Yaskawa INFORM job: R1_W49-52-A1(90,180)KM-OK.JBI

/JOB
//NAME R1_W49-52-A1(90,180)KM-OK
///FOLDERNAME KRIS-SCIANA
//POS
///NPOS 79,79,0,5,0,0
///TOOL 0
///POSTYPE PULSE
///PULSE
C00000=109471,-80411,-71829,-33263,113126,21380
C00001=-48619,-15555,-18243,-18279,95335,-12517
C00002=-74776,32390,22089,-16092,92623,-17270
C00003=-74867,35757,29537,-16050,89859,-16941
C00004=-75036,36599,32361,-16047,88568,-16832
C00005=-75036,36895,33395,-16047,88102,-16772
C00006=-74903,37254,32698,-16044,88719,-16805
C00007=-72459,12362,8558,-16008,91190,-16266
C00008=-61209,-17232,-1681,-36622,66784,-6421
C00009=-61731,-16191,-908,-36534,66611,-6591
C00010=-59990,-21702,-9204,-36261,69196,-6738
C00011=-72720,3761,1433,-15340,81732,-21663
C00012=-72610,7758,8804,-15444,79356,-21325
C00013=-73045,10828,13692,-15468,77892,-21294
C00014=-73045,10997,14245,-15480,77647,-21262
C00015=-73045,10828,13692,-15468,77892,-21294
C00016=-72048,12642,15323,-15567,78014,-20955
C00017=-73045,10828,13692,-15468,77892,-21294
C00018=-79642,10121,9779,-4752,79820,-25647
C00019=-80358,6534,2777,-4651,82236,-25983
C00020=-69953,-20577,-2415,-29105,71989,2082
C00021=-71388,-15105,4995,-29275,69960,2047
C00022=-71943,-12839,8075,-29360,69127,2048
C00023=-71949,-11985,10076,-29503,68430,2234
C00024=-71943,-12839,8075,-29360,69127,2048
C00025=-78156,-21778,1298,-21120,59983,-2481
C00026=-78744,-20042,2543,-20963,59953,-2712
C00027=-78156,-21778,1298,-21120,59983,-2481
C00028=-77865,-24315,-1842,-21059,60645,-2495
C00029=-77104,-30529,-9436,-20946,62223,-2499
C00030=-66753,-24791,-5212,-33273,69818,4262
C00031=-68453,-19258,1867,-33429,67885,4157
C00032=-69108,-16977,4805,-33509,67096,4131
C00033=-69405,-16270,5329,-33473,67016,4031
C00034=-69412,-15422,7310,-33651,66355,4242
C00035=-69405,-16270,5329,-33473,67016,4031
C00036=-69108,-16977,4805,-33509,67096,4131
C00037=-78682,-30038,-3543,-25118,55124,-1302
C00038=-79303,-28327,-2398,-24897,55100,-1566
C00039=-78682,-30038,-3543,-25118,55124,-1302
C00040=-75986,-28450,-4438,-25449,57169,-654
C00041=-75599,-31023,-7408,-25413,57744,-634
C00042=-74583,-37366,-14608,-25368,59113,-542
C00043=-54832,-34796,3895,-72693,39731,-39244
C00044=-56965,-32089,5608,-72268,38461,-39820
C00045=-57882,-31468,9455,-80412,35987,-35279
C00046=-57943,-31847,4343,-71137,38137,-40613
C00047=-56828,-32279,5486,-72299,38543,-39782
C00048=-56494,-29260,14044,-87349,37133,-31586
C00049=-56951,-32108,5596,-72272,38470,-39816
C00050=-54817,-34814,3883,-72695,39739,-39240
C00051=-70512,18761,16215,-24928,63616,-33333
C00052=-71276,21755,18910,-24702,63280,-33571
C00053=-71200,18616,16875,-24804,62971,-33467
C00054=-70825,17807,14425,-24705,64080,-33568
C00055=-67366,10962,9433,-25880,64732,-32303
C00056=-67541,9161,7476,-25769,64930,-32423
C00057=-66799,6994,5573,-25983,65214,-32188
C00058=-71450,3986,10861,-16686,71001,-58886
C00059=-83506,38901,46150,-14860,73867,-63488
C00060=-83557,40717,50113,-14966,72402,-63324
C00061=-72489,19688,28494,-17099,68495,19316
C00062=-72729,20279,28486,-17025,68740,19190
C00063=-86229,35527,44055,-7657,69598,-64559
C00064=-83557,39592,48403,-4091,67286,-63785
C00065=-82033,27096,36992,-6435,61524,-62871
C00066=-80468,765,21137,-10528,40199,-59994
C00067=-83053,-10240,21848,-3806,20837,-60444
C00068=-83052,-10243,21845,-3807,20837,-60443
C00069=-68410,-14368,18791,-25286,23146,-48376
C00070=-67879,-14666,18605,-25978,23265,-47975
C00071=-67391,-14563,19188,-26892,23140,-47472
C00072=-67758,-15818,19043,-27038,22532,-47449
C00073=-67911,-23908,2369,-21552,28082,-50172
C00074=-67911,-23908,2369,-21552,28082,-50172
C00075=-73405,-104993,-53637,-20388,20000,-51360
C00076=-27978,-168994,-134866,-21563,-5876,-50681
C00077=15433,-168994,-134866,-21563,-5876,-50681
C00078=15433,-168994,-134866,-21563,-5876,-50681
BC00000=66192,1897,868014
BC00001=55231,1826,395730
BC00002=53649,1816,327568
BC00003=53649,1816,327568
BC00004=53649,1816,327568
BC00005=53649,1816,327568
BC00006=53649,1816,327568
BC00007=53649,1816,327568
BC00008=53649,1816,327568
BC00009=53649,1816,327568
BC00010=53649,1816,327568
BC00011=81522,15,359812
BC00012=81522,15,359812
BC00013=81522,15,359812
BC00014=81522,15,359812
BC00015=81522,15,359812
BC00016=81522,15,359812
BC00017=81522,15,359812
BC00018=81522,15,359812
BC00019=81522,15,359812
BC00020=119220,15,404761
BC00021=119220,15,404761
BC00022=119220,15,404761
BC00023=119220,15,404761
BC00024=119220,15,404761
BC00025=119220,15,404761
BC00026=119220,15,404761
BC00027=119220,15,404761
BC00028=119220,15,404761
BC00029=119220,15,404761
BC00030=91379,15,388853
BC00031=91379,15,388853
BC00032=91379,15,388853
BC00033=91379,15,388853
BC00034=91379,15,388853
BC00035=91379,15,388853
BC00036=91379,15,388853
BC00037=91379,15,388853
BC00038=91379,15,388853
BC00039=91379,15,388853
BC00040=91379,15,388853
BC00041=91379,15,388853
BC00042=91379,15,388853
BC00043=52539,15,360662
BC00044=53193,15,340173
BC00045=53455,15,331978
BC00046=53455,15,331978
BC00047=53455,15,331978
BC00048=85993,15,331095
BC00049=85731,15,339290
BC00050=85076,15,359778
BC00051=28900,15,309803
BC00052=29839,15,300407
BC00053=29839,15,300407
BC00054=29839,15,300407
BC00055=36980,15,283561
BC00056=36041,15,292958
BC00057=33695,15,316449
BC00058=58127,15,406832
BC00059=58127,15,406832
BC00060=58127,15,406832
BC00061=57102,15,378985
BC00062=57102,15,378985
BC00063=58127,15,406832
BC00064=58127,15,406832
BC00065=58127,15,406832
BC00066=58127,15,406832
BC00067=58127,15,406831
BC00068=58127,15,406831
BC00069=58127,15,406831
BC00070=58127,15,406831
BC00071=58127,15,406831
BC00072=58127,15,406831
BC00073=58127,15,406831
BC00074=58127,15,406831
BC00075=58127,15,406831
BC00076=8067,559,1056049
BC00077=8067,559,1056049
BC00078=8067,551683,1056049
///POSTYPE BASE
///RECTAN
///RCONF 0,0,0,0,1,0,0,0,0,0,0,0,0,0,0,0,0,0,0,0,0,0,0,0
P00006=2.006,1.622,-0.565,0.0000,0.0000,0.0000
///RCONF 0,0,0,0,0,0,0,0,0,0,0,0,0,0,0,0,0,0,0,0,0,0,0,0
P00023=-2.957,-4.083,2.762,0.0000,0.0000,0.0000
P00024=-1.466,-0.226,-0.419,0.0000,0.0000,0.0000
P00026=2.644,0.055,-2.583,0.0000,0.0000,0.0000
P00027=2.278,0.099,-4.210,0.0000,0.0000,0.0000
//INST
///DATE 2024/09/16 12:19
///ATTR SC,RW
///GROUP1 RB1,BS1
NOP
'r1_W49-52-A1(90,180)
SFTOF
MOVJ C00000 BC00000 VJ=50.00
MOVJ C00001 BC00001 VJ=100.00
MOVJ C00002 BC00002 VJ=50.00
MOVJ C00003 BC00003 VJ=20.00
MOVL C00004 BC00004 V=60.0
REFP 3 C00005 BC00005
CALL JOB:SEARCH-R1
SET P026 P006
SFTON P026
MOVL C00006 BC00006 V=60.0
MOVL C00007 BC00007 V=100.0
MOVL C00008 BC00008 V=83.3
REFP 3 C00009 BC00009
CALL JOB:SEARCH-R1
SET P026 P006
SFTON P026
MOVL C00010 BC00010 V=60.0
'Path S1206
SFTOF
MOVJ C00011 BC00011 VJ=50.00
MOVJ C00012 BC00012 VJ=50.00
MOVL C00013 BC00013 V=60.0
REFP 3 C00014 BC00014
CALL JOB:SEARCH-R1
SET P024 P006
SFTON P024
MOVL C00015 BC00015 V=60.0
REFP 3 C00016 BC00016
CALL JOB:SEARCH-R1
SET P024 P006
SFTON P024
MOVL C00017 BC00017 V=60.0
MOVL C00018 BC00018 V=100.0
MOVL C00019 BC00019 V=166.7
'Path S1207
SFTOF
MOVJ C00020 BC00020 VJ=50.00
MOVJ C00021 BC00021 VJ=50.00
MOVL C00022 BC00022 V=60.0
REFP 3 C00023 BC00023
CALL JOB:SEARCH-R1
SET P023 P006
SFTON P023
MOVL C00024 BC00024 V=60.0
MOVL C00025 BC00025 V=60.0
REFP 3 C00026 BC00026
CALL JOB:SEARCH-R1
SET P023 P006
SFTON P023
MOVL C00027 BC00027 V=60.0
MOVL C00028 BC00028 V=100.0
MOVL C00029 BC00029 V=100.0
'Path S1208
SFTOF
MOVJ C00030 BC00030 VJ=50.00
MOVJ C00031 BC00031 VJ=50.00
MOVL C00032 BC00032 V=100.0
MOVL C00033 BC00033 V=60.0
REFP 3 C00034 BC00034
CALL JOB:SEARCH-R1
SET P027 P006
SFTON P027
MOVL C00035 BC00035 V=60.0
MOVL C00036 BC00036 V=100.0
MOVL C00037 BC00037 V=60.0
REFP 3 C00038 BC00038
CALL JOB:SEARCH-R1
SET P027 P006
SFTON P027
MOVL C00039 BC00039 V=60.0
MOVL C00040 BC00040 V=100.0
MOVL C00041 BC00041 V=100.0
MOVL C00042 BC00042 V=166.7
'Path W1209
SFTOF
SFTON P027
CALL JOB:COFNIJ_DRUT
MOVJ C00043 BC00043 VJ=20.00
MOVJ C00044 BC00044 VJ=20.00
MOVL C00045 BC00045 V=100.0 PL=0
REFP 1 C00046 BC00046
REFP 2 C00047 BC00047
MACRO1 MJ#(0) ARGF7
SFTON P023
ARCON
MOVL C00048 BC00048 V=7.5
ARCOF
MOVL C00049 BC00049 V=166.7
MOVL C00050 BC00050 V=166.7
SFTOF
'Path W1210
SFTOF
SFTON P024
MOVJ C00051 BC00051 VJ=20.00
MOVL C00052 BC00052 V=100.0 PL=0
REFP 1 C00053 BC00053
REFP 2 C00054 BC00054
MACRO1 MJ#(0) ARGF6
ARCON
WVON WEV#(40)
MOVL C00055 BC00055 V=7.5
ARCOF
WVOF
MOVL C00056 BC00056 V=166.7
MOVL C00057 BC00057 V=166.7
SFTOF
'Path W1212
SFTOF
SFTON P026
MOVJ C00058 BC00058 VJ=20.00
MOVJ C00059 BC00059 VJ=20.00
MOVL C00060 BC00060 V=100.0 PL=0
REFP 1 C00061 BC00061
REFP 2 C00062 BC00062
MACRO1 MJ#(0) ARGF9
ARCON
MOVL C00063 BC00063 V=10.0
MOVL C00064 BC00064 V=10.0
MOVL C00065 BC00065 V=10.8
SFTON P024
MOVL C00066 BC00066 V=10.8
ARCON
MOVL C00067 BC00067 V=10.8
MOVL C00068 BC00068 V=10.3
MOVL C00069 BC00069 V=10.3
MOVL C00070 BC00070 V=10.3
MOVL C00071 BC00071 V=10.3
MOVL C00072 BC00072 V=10.3
ARCOF
MOVL C00073 BC00073 V=166.7
MOVL C00074 BC00074 V=166.7
SFTOF
MOVJ C00075 BC00075 VJ=100.00
MOVJ C00076 BC00076 VJ=100.00
MOVJ C00077 BC00077 VJ=100.00
MOVJ C00078 BC00078 VJ=100.00
END
